# EPICS autosave request: iocBoot/iocmw100ex/mw100_labels.req
$(P)$(DAU):001:Label
$(P)$(DAU):002:Label
$(P)$(DAU):003:Label
$(P)$(DAU):004:Label
$(P)$(DAU):005:Label
$(P)$(DAU):006:Label
$(P)$(DAU):007:Label
$(P)$(DAU):008:Label
$(P)$(DAU):009:Label
$(P)$(DAU):010:Label

$(P)$(DAU):011:Label
$(P)$(DAU):012:Label
$(P)$(DAU):013:Label
$(P)$(DAU):014:Label
$(P)$(DAU):015:Label
$(P)$(DAU):016:Label
$(P)$(DAU):017:Label
$(P)$(DAU):018:Label
#$(P)$(DAU):019:Label
#$(P)$(DAU):020:Label

$(P)$(DAU):021:Label
$(P)$(DAU):022:Label
$(P)$(DAU):023:Label
$(P)$(DAU):024:Label
$(P)$(DAU):025:Label
$(P)$(DAU):026:Label
$(P)$(DAU):027:Label
$(P)$(DAU):028:Label
$(P)$(DAU):029:Label
$(P)$(DAU):030:Label

#$(P)$(DAU):031:Label
#$(P)$(DAU):032:Label
#$(P)$(DAU):033:Label
#$(P)$(DAU):034:Label
#$(P)$(DAU):035:Label
#$(P)$(DAU):036:Label
#$(P)$(DAU):037:Label
#$(P)$(DAU):038:Label
#$(P)$(DAU):039:Label
#$(P)$(DAU):040:Label

#$(P)$(DAU):041:Label
#$(P)$(DAU):042:Label
#$(P)$(DAU):043:Label
#$(P)$(DAU):044:Label
#$(P)$(DAU):045:Label
#$(P)$(DAU):046:Label
#$(P)$(DAU):047:Label
#$(P)$(DAU):048:Label
#$(P)$(DAU):049:Label
#$(P)$(DAU):050:Label

#$(P)$(DAU):051:Label
#$(P)$(DAU):052:Label
#$(P)$(DAU):053:Label
#$(P)$(DAU):054:Label
#$(P)$(DAU):055:Label
#$(P)$(DAU):056:Label
#$(P)$(DAU):057:Label
#$(P)$(DAU):058:Label
#$(P)$(DAU):059:Label
#$(P)$(DAU):060:Label

$(P)$(DAU):C001:Label
$(P)$(DAU):C002:Label
$(P)$(DAU):C003:Label
$(P)$(DAU):C004:Label
$(P)$(DAU):C005:Label
$(P)$(DAU):C006:Label
$(P)$(DAU):C007:Label
$(P)$(DAU):C008:Label
$(P)$(DAU):C009:Label
$(P)$(DAU):C010:Label

$(P)$(DAU):A001:Label
$(P)$(DAU):A002:Label
$(P)$(DAU):A003:Label
$(P)$(DAU):A004:Label
$(P)$(DAU):A005:Label
$(P)$(DAU):A006:Label
$(P)$(DAU):A007:Label
$(P)$(DAU):A008:Label
$(P)$(DAU):A009:Label
$(P)$(DAU):A010:Label
$(P)$(DAU):A011:Label
$(P)$(DAU):A012:Label
$(P)$(DAU):A013:Label
$(P)$(DAU):A014:Label
$(P)$(DAU):A015:Label
$(P)$(DAU):A016:Label
$(P)$(DAU):A017:Label
$(P)$(DAU):A018:Label
$(P)$(DAU):A019:Label
$(P)$(DAU):A020:Label
$(P)$(DAU):A021:Label
$(P)$(DAU):A022:Label
$(P)$(DAU):A023:Label
$(P)$(DAU):A024:Label
$(P)$(DAU):A025:Label
$(P)$(DAU):A026:Label
$(P)$(DAU):A027:Label
$(P)$(DAU):A028:Label
$(P)$(DAU):A029:Label
$(P)$(DAU):A030:Label
$(P)$(DAU):A031:Label
$(P)$(DAU):A032:Label
$(P)$(DAU):A033:Label
$(P)$(DAU):A034:Label
$(P)$(DAU):A035:Label
$(P)$(DAU):A036:Label
$(P)$(DAU):A037:Label
$(P)$(DAU):A038:Label
$(P)$(DAU):A039:Label
$(P)$(DAU):A040:Label
$(P)$(DAU):A041:Label
$(P)$(DAU):A042:Label
$(P)$(DAU):A043:Label
$(P)$(DAU):A044:Label
$(P)$(DAU):A045:Label
$(P)$(DAU):A046:Label
$(P)$(DAU):A047:Label
$(P)$(DAU):A048:Label
$(P)$(DAU):A049:Label
$(P)$(DAU):A050:Label
$(P)$(DAU):A051:Label
$(P)$(DAU):A052:Label
$(P)$(DAU):A053:Label
$(P)$(DAU):A054:Label
$(P)$(DAU):A055:Label
$(P)$(DAU):A056:Label
$(P)$(DAU):A057:Label
$(P)$(DAU):A058:Label
$(P)$(DAU):A059:Label
$(P)$(DAU):A060:Label

$(P)$(DAU):K001:Label
$(P)$(DAU):K002:Label
$(P)$(DAU):K003:Label
$(P)$(DAU):K004:Label
$(P)$(DAU):K005:Label
$(P)$(DAU):K006:Label
$(P)$(DAU):K007:Label
$(P)$(DAU):K008:Label
$(P)$(DAU):K009:Label
$(P)$(DAU):K010:Label
